// TIA Portal V21 export
// export: Created 2000-01-01T00:00:00.0000000Z, ExportSetting None
ORGANIZATION_BLOCK "Cyclic_Main"   // OB200, SCL, ProgramCycle
{ S7_Optimized_Access := 'TRUE' }
// 主程序循环 OB1（梯形图）。每个扫描周期调用一次 FC_StartStop 处理起保停逻辑。
// stored: SetENOAutomatically false
   VAR_INPUT
      Initial_Call : Bool;
      Remanence : Bool;
   END_VAR
BEGIN
// 调用起保停 FC
// 调用起保停功能：FC_StartStop 内部读 I_Start/I_Stop/I_EStop，写 Q_Run
   "FC_StartStop"();
END_ORGANIZATION_BLOCK
